// TwinCAT 3 PLC project Untitled1
// ProgramVersion: 3.1.0.8
// libraries:
//   Tc2_Standard, * (Beckhoff Automation GmbH)
//   Tc2_System, * (Beckhoff Automation GmbH)
//   Tc3_Interfaces, * (Beckhoff Automation GmbH)
//   Tc3_Module, * (Beckhoff Automation GmbH)
//   Tc3_PLCopen_OpcUa, * (Beckhoff Automation GmbH)
// project tree:
//   DUTs/ManualModule/ DUT_MANUALMODULE_PARAMETER.TcDUT, DUT_MANUALMODULE.TcDUT
//   DUTs/MessageFeed/ DUT_MESSAGEFEED.TcDUT
//   DUTs/Module Interface/ DUT_MODULE_INTERFACE.TcDUT
//   DUTs/Module Interface/Input/ DUT_MODE.TcDUT, DUT_MODULE_INTERFACE_INPUT.TcDUT, DUT_PARAMETER_INPUT.TcDUT, DUT_SKILL_INPUT.TcDUT
//   DUTs/Module Interface/Output/ DUT_MODULE_INTERFACE_OUTPUT.TcDUT, DUT_PARAMETER_OUTPUT.TcDUT, DUT_SKILL_OUTPUT.TcDUT, DUT_STATEVALUES.TcDUT
//   DUTs/Production List/ DUT_PARAMETER.TcDUT, DUT_SKILL.TcDUT, DUT_TASK.TcDUT, DUT_TASKSTATE.TcDUT
//   DUTs/Queue/ DUT_RECIPEORDER.TcDUT, DUT_RECIPE_USERPARAMETERINPUT.TcDUT
//   DUTs/RecipeOffer/ DUT_RECIPE_OFFER.TcDUT, DUT_RECIPE_USERPARAMETEROUTPUT.TcDUT
//   DUTs/Server DUTs/ DUT_SERVER_MODULE_INTERFACE.TcDUT, DUT_SERVER_MODULE_INTERFACE_INPUT.TcDUT, DUT_SERVER_MODULE_INTERFACE_OUTPUT.TcDUT, DUT_SERVER_PARAMETERINPUTARRAY.TcDUT, DUT_SERVER_PARAMETEROUTPUTARRAY.TcDUT, DUT_SERVER_SKILLINPUTARRAY.TcDUT, DUT_SERVER_SKILLOUTPUTARRAY.TcDUT, DUT_SERVER_SKILL_INPUT.TcDUT, DUT_SERVER_SKILL_OUTPUT.TcDUT, DUT_SERVER_STATEVALUEARRAY.TcDUT
//   GVLs/ MI5.TcGVL, OpcServerConstants.TcGVL
//   / PlcTask.TcTTO
//   POUs/FakeHandModule/ FB_Fake2401.TcPOU
//   POUs/ MAIN.TcPOU
// real-time tasks:
//   TASK PlcTask: cycle T#5ms, priority 4, ADS port 350

CONFIGURATION Untitled1
    RESOURCE PLC ON TwinCAT3
        TASK PlcTask(INTERVAL := T#5ms, PRIORITY := 4);
        PROGRAM MAIN WITH PlcTask : MAIN;
    END_RESOURCE
END_CONFIGURATION

// ---- DUTs/ManualModule/DUT_MANUALMODULE_PARAMETER.TcDUT
TYPE DUT_MANUALMODULE_PARAMETER :
STRUCT
	Name: STRING(80);
	ID: UINT;
	Unit: STRING(80);
	Value: LREAL;
	StringValue: STRING(80);
END_STRUCT
END_TYPE

// ---- DUTs/ManualModule/DUT_MANUALMODULE.TcDUT
TYPE DUT_MANUALMODULE :
STRUCT
	SkillDescription: STRING(80);
	SkillID: UINT;
	TaskID: UINT;
	Ready: BOOL;
	Busy: BOOL;
	Done: BOOL;
	Execute: BOOL;
	Error: BOOL;
	ErrorID: UINT;
	Position: LREAL;
	Parameter: ARRAY[0..ParameterCnt] OF DUT_MANUALMODULE_PARAMETER;
END_STRUCT
END_TYPE

// ---- DUTs/MessageFeed/DUT_MESSAGEFEED.TcDUT
TYPE DUT_MESSAGEFEED :
STRUCT
	ID: INT;
	Level: INT; //1:Success; 2:Info; 3:Warning; 4:ERROR; 5:FATAL
	Timestamp: STRING[80];
	Message: STRING[256];
END_STRUCT
END_TYPE

// ---- DUTs/Module Interface/DUT_MODULE_INTERFACE.TcDUT
/// MODULE INTERFACE INPUT AND OUTPUT 
TYPE DUT_MODULE_INTERFACE :
STRUCT
	///Information that the module reads
	Input: DUT_MODULE_INTERFACE_INPUT;
	///Information that the module write
	Output: DUT_MODULE_INTERFACE_OUTPUT;
END_STRUCT
END_TYPE

// ---- DUTs/Module Interface/Input/DUT_MODE.TcDUT
/// MODE to run (inside of MODULE_INTERFACE_INPUT)
TYPE DUT_MODE :
(
	///Initialitzation number mode
	Init := 0,
	///Automatic number mode
	Auto := 1,
	///Manual number mode
	Manual := 2,
	Reset := 3
);
END_TYPE

// ---- DUTs/Module Interface/Input/DUT_MODULE_INTERFACE_INPUT.TcDUT
TYPE DUT_MODULE_INTERFACE_INPUT :
STRUCT
	///Mode to run (init,auto,manual,..)
	Mode: DUT_MODE;
	///check if the modules is alive
	ConnectionTestInput: BOOL;
	///Modules get their position
	PositionInput: LREAL;
	///Update data= TRUE, No updatedata=FALSE
	Watchbit: BOOL;
	///Emergency stop
	EmergencyStop: BOOL;
	///Range of INPUT skills
	SkillInput: ARRAY[0..SkillCnt] OF DUT_SKILL_INPUT;
END_STRUCT
END_TYPE

// ---- DUTs/Module Interface/Input/DUT_PARAMETER_INPUT.TcDUT
TYPE DUT_PARAMETER_INPUT :
STRUCT
	///Value of the parameter 
	Value: LREAL;
	///Possibility to a string value depending on the parameter
	StringValue: STRING[80];
END_STRUCT
END_TYPE

// ---- DUTs/Module Interface/Input/DUT_SKILL_INPUT.TcDUT
TYPE DUT_SKILL_INPUT :
STRUCT
	///Range of parameters
	ParameterInput: ARRAY[0..ParameterCnt] OF DUT_PARAMETER_INPUT;
	///Start process
	Execute: BOOL;
END_STRUCT
END_TYPE

// ---- DUTs/Module Interface/Output/DUT_MODULE_INTERFACE_OUTPUT.TcDUT
TYPE DUT_MODULE_INTERFACE_OUTPUT :
STRUCT
	///Free to use = TRUE, busy to use =FALSE
	Dummy: BOOL := TRUE;
	///Individual name of the module
	Name: STRING(80);
	///Identification number of module
	ID: UINT;
	///IP address
	IP: STRING(80);
	///Show if the module is in Standby or not
	Idle: BOOL;
	///Show if the module is connected
	Connected: BOOL;
	///Feedback with conection test input
	ConnectionTestOutput: BOOL;
	///Show if the system has error when=TRUE
	Error: BOOL;
	///Identification number of the error
	ErrorID: UINT;
	///Description of the error
	ErrorDescription: STRING(80);
	///Description of the current task
	CurrentTaskDescription: STRING(80);
	
	PositionOutput	: LREAL; //actual position of the modules, calculated by the module itself
	///Position of the sensor
	PositionSensor: BOOL;
	///Range of OUTPUT skills
	SkillOutput: ARRAY[0..SkillCnt] OF DUT_SKILL_OUTPUT;
	///Range of state values
	StateValue: ARRAY[0..StateCnt] OF DUT_STATEVALUES;
END_STRUCT
END_TYPE

// ---- DUTs/Module Interface/Output/DUT_PARAMETER_OUTPUT.TcDUT
TYPE DUT_PARAMETER_OUTPUT :
STRUCT
	///Free to use = TRUE, busy to use =FALSE
	Dummy: BOOL := TRUE;
	///ID of the parameter
	ID: UINT;
	///Name of the parameter
	Name: STRING[80];
	///Unit of the parameter
	Unit: STRING[80];
	///Optional parameter
	Required: BOOL;
	///Default parameter to work
	Default: LREAL;
	///Minimum value of the parameter
	MinValue: LREAL;
	///Maximum value of the parameter
	MaxValue: LREAL;
END_STRUCT
END_TYPE

// ---- DUTs/Module Interface/Output/DUT_SKILL_OUTPUT.TcDUT
TYPE DUT_SKILL_OUTPUT :
STRUCT
	//Free to use = TRUE, busy to use =FALSE
	Dummy: BOOL := TRUE;
	//Identification number of skill
	ID: UINT;
	//indentfication name of skill
	Name: STRING(80);
	//Skill activated
	Activated: BOOL;
	//Ready to do skill
	Ready: BOOL;
	//Skill in process
	Busy: BOOL;
	//Skill finish
	Done: BOOL;
	//Error in system
	Error: BOOL;
	//Range of parameters
	ParameterOutput: ARRAY[0..ParameterCnt] OF DUT_PARAMETER_OUTPUT;
END_STRUCT
END_TYPE

// ---- DUTs/Module Interface/Output/DUT_STATEVALUES.TcDUT
TYPE DUT_STATEVALUES :
STRUCT
	Dummy:			BOOL := TRUE;				(*Free to use = TRUE, busy to use =FALSE*)
	Value:			LREAL;						(*Value of the State*)
	Name:			STRING[80];						(*Name of the state*)
	Description:	STRING[80];				(*Description of the state*)
	Unit:			STRING[80];						(*Unit of the state ()*)
END_STRUCT
END_TYPE

// ---- DUTs/Production List/DUT_PARAMETER.TcDUT
TYPE DUT_PARAMETER :
STRUCT
	///Free to use = TRUE, busy to use =FALSE
	Dummy: BOOL := TRUE;
	///ID of the parameter
	ID: UINT;
	///Name of the parameter
	Name: STRING[80];
	///Unit of the parameter (mm,L,...)
	Unit: STRING[80];
	///Optional parameter
	Required: BOOL;
	///Default parameter to work
	Default: LREAL;
	///Minimum value of the parameter
	MinValue: LREAL;
	///Maximum value of the parameter
	MaxValue: LREAL;
	///Actual Value
	Value: LREAL;
	///StringValue
	StringValue: STRING[80];
END_STRUCT
END_TYPE

// ---- DUTs/Production List/DUT_SKILL.TcDUT
///  Skill variables inside DUT_TASK
TYPE DUT_SKILL :
STRUCT
	///Name assigned for the process tool
	AssignedModuleName: STRING[80];
	///ID assigned for the process tool
	AssignedModuleID: UINT;
	///Position assigned for the process tool
	AssignedModulePosition: LREAL;
	///Free to use = TRUE, busy to use =FALSE
	Dummy: BOOL := TRUE;
	///Identification number of the skill
	ID: UINT;
	///Name of the skill
	Name: STRING[80];
	// State of the skill
	State: INT;
	///Range of parameters
	Parameter: ARRAY[0..ParameterCnt] OF DUT_PARAMETER;
END_STRUCT
END_TYPE

// ---- DUTs/Production List/DUT_TASK.TcDUT
TYPE DUT_TASK :
STRUCT
	///Name of the Task
	Name: STRING[80];
	///Free to use = TRUE, busy to use =FALSE
	Dummy: BOOL := TRUE;
	///Identification number of the Task
	TaskID: INT;
	///Identification number of the Recipe
	RecipeID: INT;
	///Range of Skill in the TASK
	Skill: ARRAY[0..TaskSkillCnt] OF DUT_SKILL;
	///When occurs the action
	Timestamp: STRING[80];
	///State of the TASK e.g (unassigned, assigned, waitingForSkillReady, inProgress, done, aborted, error)
	State: DUT_TASKSTATE;
	//
	AbortTask : BOOL := FALSE;
END_STRUCT
END_TYPE

// ---- DUTs/Production List/DUT_TASKSTATE.TcDUT
TYPE DUT_TASKSTATE :
(
	Unassigned := 0,
	//Assigned := 1,
	WaitingForSkillReady := 1,
	InProgress := 2,
	Done := 3,
	Aborted := 4,
	Error := 5
);
END_TYPE

// ---- DUTs/Queue/DUT_RECIPEORDER.TcDUT
TYPE DUT_RECIPEORDER :
STRUCT
	Locked	: BOOL;
	Pending: BOOL;
	///corelating to the offered recipes#
	RecipeID: INT;
	///continious numbering
	TaskID: INT;
	Name	: STRING[80];
	Description: STRING[255];
	UserParameter: ARRAY [0..UserParameterCnt] OF DUT_RECIPE_USERPARAMETERINPUT;
END_STRUCT
END_TYPE

// ---- DUTs/Queue/DUT_RECIPE_USERPARAMETERINPUT.TcDUT
TYPE DUT_RECIPE_USERPARAMETERINPUT :
STRUCT
	Value: REAL;
END_STRUCT
END_TYPE

// ---- DUTs/RecipeOffer/DUT_RECIPE_OFFER.TcDUT
TYPE DUT_RECIPE_OFFER :
STRUCT
	Dummy:			BOOL := TRUE;
	Name:			STRING[80]:= 'e.g. Product x';
	RecipeID:		INT;
	Description:	STRING[255]:= '%Description of the Recipe e.g. "a recipe, that produces a product with feature x"';
	UserParameter:  ARRAY [0..UserParameterCnt] OF DUT_RECIPE_USERPARAMETEROUTPUT;
END_STRUCT
END_TYPE

// ---- DUTs/RecipeOffer/DUT_RECIPE_USERPARAMETEROUTPUT.TcDUT
TYPE DUT_RECIPE_USERPARAMETEROUTPUT :
STRUCT
	Dummy:			BOOL := TRUE;
	Name:			STRING[80];
	Description:	STRING[80];
	Unit:			STRING[80];
	MinValue:		LREAL;
	MaxValue:		LREAL;
	Default:		LREAL;
	Step:			LREAL;
END_STRUCT
END_TYPE

// ---- DUTs/Server DUTs/DUT_SERVER_MODULE_INTERFACE.TcDUT
/// MODULE INTERFACE INPUT AND OUTPUT 
TYPE DUT_SERVER_MODULE_INTERFACE :
STRUCT
	///Information that the module reads
	Input: DUT_SERVER_MODULE_INTERFACE_INPUT;
	///Information that the module write
	Output: DUT_SERVER_MODULE_INTERFACE_OUTPUT;
END_STRUCT
END_TYPE

// ---- DUTs/Server DUTs/DUT_SERVER_MODULE_INTERFACE_INPUT.TcDUT
TYPE DUT_SERVER_MODULE_INTERFACE_INPUT :
STRUCT
	///Mode to run (init,auto,manual,..)
	Mode: INT;
	///check if the modules is alive
	ConnectionTestInput: BOOL;
	///Modules get their position
	PositionInput: LREAL;
	///Update data= TRUE, No updatedata=FALSE
	Watchbit: BOOL;
	///Emergency stop
	EmergencyStop: BOOL;
	///Range of INPUT skills
	SkillInput: DUT_SERVER_SKILLINPUTARRAY;
END_STRUCT
END_TYPE

// ---- DUTs/Server DUTs/DUT_SERVER_MODULE_INTERFACE_OUTPUT.TcDUT
TYPE DUT_SERVER_MODULE_INTERFACE_OUTPUT :
STRUCT
	///Free to use = TRUE, busy to use =FALSE
	Dummy: BOOL := TRUE;
	///Individual name of the module
	Name: STRING(80);
	///Identification number of module
	ID: UINT;
	///IP address
	IP: STRING(80);
	///Show if the module is in Standby or not
	Idle: BOOL;
	///Show if the module is connected
	Connected: BOOL;
	///Feedback with conection test input
	ConnectionTestOutput: BOOL;
	///Show if the system has error when=TRUE
	Error: BOOL;
	///Identification number of the error
	ErrorID: UINT;
	///Description of the error
	ErrorDescription: STRING(80);
	///Description of the current task
	CurrentTaskDescription: STRING(80);
	///Position of the output
	PositionOutput: LREAL;
	/// Bool value of the Sensor
	PositionSensor: BOOL;
	///Range of OUTPUT skills
	SkillOutput: DUT_SERVER_SKILLOUTPUTARRAY;
	///Range of state values
	StateValue: DUT_SERVER_STATEVALUEARRAY;
END_STRUCT
END_TYPE

// ---- DUTs/Server DUTs/DUT_SERVER_PARAMETERINPUTARRAY.TcDUT
TYPE DUT_SERVER_PARAMETERINPUTARRAY :
STRUCT
	ParameterInput0: DUT_PARAMETER_INPUT;
	ParameterInput1: DUT_PARAMETER_INPUT;
	ParameterInput2: DUT_PARAMETER_INPUT;
	ParameterInput3: DUT_PARAMETER_INPUT;
	ParameterInput4: DUT_PARAMETER_INPUT;
	ParameterInput5: DUT_PARAMETER_INPUT;
END_STRUCT
END_TYPE

// ---- DUTs/Server DUTs/DUT_SERVER_PARAMETEROUTPUTARRAY.TcDUT
TYPE DUT_SERVER_PARAMETEROUTPUTARRAY :
STRUCT
	ParameterOutput0: DUT_PARAMETER_OUTPUT;
	ParameterOutput1: DUT_PARAMETER_OUTPUT;
	ParameterOutput2: DUT_PARAMETER_OUTPUT;
	ParameterOutput3: DUT_PARAMETER_OUTPUT;
	ParameterOutput4: DUT_PARAMETER_OUTPUT;
	ParameterOutput5: DUT_PARAMETER_OUTPUT;
END_STRUCT
END_TYPE

// ---- DUTs/Server DUTs/DUT_SERVER_SKILLINPUTARRAY.TcDUT
TYPE DUT_SERVER_SKILLINPUTARRAY :
STRUCT
	SkillInput0: DUT_SERVER_SKILL_INPUT;
	SkillInput1: DUT_SERVER_SKILL_INPUT;
	SkillInput2: DUT_SERVER_SKILL_INPUT;
	SkillInput3: DUT_SERVER_SKILL_INPUT;
	SkillInput4: DUT_SERVER_SKILL_INPUT;
	SkillInput5: DUT_SERVER_SKILL_INPUT;
	SkillInput6: DUT_SERVER_SKILL_INPUT;
	SkillInput7: DUT_SERVER_SKILL_INPUT;
	SkillInput8: DUT_SERVER_SKILL_INPUT;
	SkillInput9: DUT_SERVER_SKILL_INPUT;
	SkillInput10: DUT_SERVER_SKILL_INPUT;
	SkillInput11: DUT_SERVER_SKILL_INPUT;
	SkillInput12: DUT_SERVER_SKILL_INPUT;
	SkillInput13: DUT_SERVER_SKILL_INPUT;
	SkillInput14: DUT_SERVER_SKILL_INPUT;
	SkillInput15: DUT_SERVER_SKILL_INPUT;
END_STRUCT
END_TYPE

// ---- DUTs/Server DUTs/DUT_SERVER_SKILLOUTPUTARRAY.TcDUT
TYPE DUT_SERVER_SKILLOUTPUTARRAY :
STRUCT
	SkillOutput0: DUT_SERVER_SKILL_OUTPUT;
	SkillOutput1: DUT_SERVER_SKILL_OUTPUT;
	SkillOutput2: DUT_SERVER_SKILL_OUTPUT;
	SkillOutput3: DUT_SERVER_SKILL_OUTPUT;
	SkillOutput4: DUT_SERVER_SKILL_OUTPUT;
	SkillOutput5: DUT_SERVER_SKILL_OUTPUT;
	SkillOutput6: DUT_SERVER_SKILL_OUTPUT;
	SkillOutput7: DUT_SERVER_SKILL_OUTPUT;
	SkillOutput8: DUT_SERVER_SKILL_OUTPUT;
	SkillOutput9: DUT_SERVER_SKILL_OUTPUT;
	SkillOutput10: DUT_SERVER_SKILL_OUTPUT;
	SkillOutput11: DUT_SERVER_SKILL_OUTPUT;
	SkillOutput12: DUT_SERVER_SKILL_OUTPUT;
	SkillOutput13: DUT_SERVER_SKILL_OUTPUT;
	SkillOutput14: DUT_SERVER_SKILL_OUTPUT;
	SkillOutput15: DUT_SERVER_SKILL_OUTPUT;
END_STRUCT
END_TYPE

// ---- DUTs/Server DUTs/DUT_SERVER_SKILL_INPUT.TcDUT
TYPE DUT_SERVER_SKILL_INPUT :
STRUCT
	///Range of parameters
	ParameterInput: DUT_SERVER_PARAMETERINPUTARRAY;
	///Start process
	Execute: BOOL;
END_STRUCT
END_TYPE

// ---- DUTs/Server DUTs/DUT_SERVER_SKILL_OUTPUT.TcDUT
TYPE DUT_SERVER_SKILL_OUTPUT :
STRUCT
	///Free to use = TRUE, busy to use =FALSE
	Dummy: BOOL := TRUE;
	///Identification number of skill
	ID: UINT;
	///indentfication name of skill
	Name: STRING(80);
	///Skill activated
	Activated: BOOL;
	///Ready to do skill
	Ready: BOOL;
	///Skill in process
	Busy: BOOL;
	///Skill finish
	Done: BOOL;
	///Error in system
	Error: BOOL;
	///Range of parameters
	ParameterOutput: DUT_SERVER_PARAMETEROUTPUTARRAY;
END_STRUCT
END_TYPE

// ---- DUTs/Server DUTs/DUT_SERVER_STATEVALUEARRAY.TcDUT
TYPE DUT_SERVER_STATEVALUEARRAY :
STRUCT
	StateValue0: DUT_STATEVALUES;
	StateValue1: DUT_STATEVALUES;
	StateValue2: DUT_STATEVALUES;
	StateValue3: DUT_STATEVALUES;
	StateValue4: DUT_STATEVALUES;
	StateValue5: DUT_STATEVALUES;
	StateValue6: DUT_STATEVALUES;
	StateValue7: DUT_STATEVALUES;
	StateValue8: DUT_STATEVALUES;
	StateValue9: DUT_STATEVALUES;
	StateValue10: DUT_STATEVALUES;
END_STRUCT
END_TYPE

// ---- GVLs/MI5.TcGVL
VAR_GLOBAL
	(*{attribute 'OPC.UA.DA' := '1'}
	oldModule2401 : DUT_SERVER_MODULE_INTERFACE;
		{attribute 'OPC.UA.DA' := '1'}
	oldModule2402 : DUT_SERVER_MODULE_INTERFACE;
	{attribute 'OPC.UA.DA' := '1'}
	oldProductionList		: ARRAY [0..TaskCnt] OF DUT_SERVER_TASK;
	{attribute 'OPC.UA.DA' := '1'}
	oldRecipe			: ARRAY [0..OfferCnt] OF DUT_RECIPEOFFER;
	{attribute 'OPC.UA.DA' := '1'}
	oldOrder			: ARRAY [0..OrderCnt] OF DUT_RECIPEORDER;
	*)
	{attribute 'OPC.UA.DA' := '1'}
	ProductionList	: ARRAY [0..TaskCnt] OF DUT_TASK;
	{attribute 'OPC.UA.DA' := '1'}
	Recipe			: ARRAY [0..OfferCnt] OF DUT_RECIPE_OFFER;
	{attribute 'OPC.UA.DA' := '1'}
	Order			: ARRAY [0..OrderCnt] OF DUT_RECIPEORDER;
		{attribute 'OPC.UA.DA' := '1'}
	MessageFeed		: ARRAY [0..MessagefeedCnt] OF DUT_MESSAGEFEED;
			{attribute 'OPC.UA.DA' := '1'}
	Module2401Manual	: DUT_MANUALMODULE;
				{attribute 'OPC.UA.DA' := '1'}
	Module2402Manual	: DUT_MANUALMODULE;
				{attribute 'OPC.UA.DA' := '1'}
	Module2403Manual	: DUT_MANUALMODULE;
	{attribute 'OPC.UA.DA' := '1'}
	Module2501			: DUT_SERVER_MODULE_INTERFACE;
	{attribute 'OPC.UA.DA' := '1'}
	Module2601			: DUT_SERVER_MODULE_INTERFACE;
END_VAR

// ---- GVLs/OpcServerConstants.TcGVL
VAR_GLOBAL CONSTANT
	
	ParameterCnt 	: INT := 5;					(*Maximum number of skillparameters*)
	SkillCnt		: INT := 15;				(*Maximum number of skills per Module*)
	StateCnt		: INT := 10;				(*Maximum number of Statevalues of one Module*)
	ModuleCnt		: INT := 10;				(*Maximum number of modules*)
	TaskCnt			: INT := 30;				(*Maximum number of Tasks in Production List*)
	OfferCnt		: INT := 30;                 (*Maximum number  *)   
	OrderCnt		: INT := 5;                       
	UserParameterCnt: INT := 5;					(*Number of user set parameters per recipe*)
	TaskSkillCnt	: INT := 50;				(*Number of skills per task*)
	MessagefeedCnt  : INT := 100;
	
END_VAR

// ---- POUs/MAIN.TcPOU
PROGRAM MAIN
VAR
	sizeOfTask : INT;
	sizeOfRecipeOffer : INT;
	sizeOfRecipeOrder: INT;
	simulateHandModule	: FB_Fake2401;
END_VAR

//OPCMODULE[1].Input.ConnectionTestInput:= OPCModule[1].Output.ConnectionTestOutput;
sizeOfTask := SIZEOF(MI5.ProductionList[0]);
sizeOfRecipeOffer := SIZEOF(MI5.Recipe[0]);
sizeOfRecipeOrder := SIZEOF(MI5.Order[0]);

simulateHandModule(position := 202.2, ManualModule := Module2401Manual);

END_PROGRAM

// ---- POUs/FakeHandModule/FB_Fake2401.TcPOU
FUNCTION_BLOCK FB_Fake2401
VAR_INPUT
	execute	: BOOL := TRUE;
	position	: LREAL := 202.02;
	Autotime	: TIME := T#5S;
END_VAR
VAR_IN_OUT
	ManualModule	: DUT_MANUALMODULE;
END_VAR
VAR_OUTPUT
END_VAR
VAR
	Autotimer	: TON;
	state : INT;
	
	userexecute		: BOOL;
	userdone		: BOOL;
	UserSkillName	: STRING[80];
	
END_VAR

IF execute THEN
	
	CASE state OF
		
	0: 
		
		ManualModule.Error 		:= FALSE;
		ManualModule.Position 	:= position;
		ManualModule.Done		:= FALSE;
		ManualModule.Ready		:= TRUE;
		
		IF ManualModule.Execute THEN
			state := 10;
			ManualModule.Ready		:= FALSE;
			ManualModule.Busy		:= TRUE;
			Autotimer(IN := FALSE);
		END_IF
		
	10: Autotimer(IN := TRUE, PT := Autotime);
		IF Autotimer.Q THEN
			userdone := TRUE;
		END_IF
		userexecute := TRUE;
		userskillname := ManualModule.SkillDescription;
		IF userdone THEN
			ManualModule.Done := TRUE;
			ManualModule.busy := FALSE;
			state := 20;
		END_IF
		
	20:
		IF NOT ManualModule.Execute THEN
			state := 0;
			userdone := FALSE;
			ManualModule.Done := FALSE;
		END_IF
	
	
	
	
	
	END_CASE
END_IF

END_FUNCTION_BLOCK
